// TIA Portal V17 export
// export: Created 2024-09-27T19:06:40.5718073Z, ExportSetting WithDefaults, DisplayName Totally Integrated Automation Portal, DisplayVersion V17, DisplayName TIA Portal Openness, DisplayVersion V17, DisplayName TIA Portal Version Control Interface, DisplayVersion V17, DisplayName STEP 7 Professional, DisplayVersion V17, DisplayName STEP 7 Safety, DisplayVersion V17, DisplayName WinCC Professional, DisplayVersion V17
ORGANIZATION_BLOCK "Main"   // OB1, LAD, ProgramCycle
TITLE = "Main Program Sweep (Cycle)"
{ S7_Optimized_Access := 'TRUE' }
VERSION : 0.1
// stored: AutoNumber true, IsIECCheckEnabled false, SetENOAutomatically false
   VAR_INPUT
      Initial_Call : Bool;   // Initial call of this OB
      Remanence : Bool;   // =True, if remanent data are available
   END_VAR
BEGIN

REGION Network 1: AUTO MODE SET FROM HMI
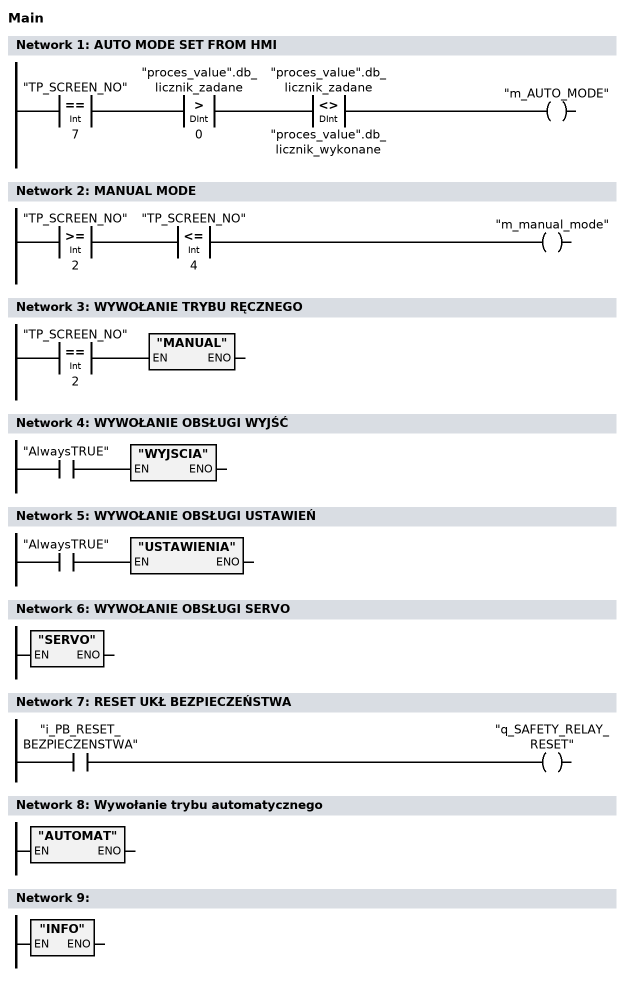
   RUNG wire#powerrail
      { S7_Templates := "SrcType := Int" } EQ_Contact(in1 := "TP_SCREEN_NO", in2 := 7)
      { S7_Templates := "SrcType := DInt" } GT_Contact(in1 := "proces_value".db_licznik_zadane, in2 := 0)
      { S7_Templates := "SrcType := DInt" } NE_Contact(in1 := "proces_value".db_licznik_zadane, in2 := "proces_value".db_licznik_wykonane)
      Coil( "m_AUTO_MODE" )
   END_RUNG
   // the same network as SCL:
   "m_AUTO_MODE" := ("TP_SCREEN_NO" = 7) AND ("proces_value".db_licznik_zadane > 0) AND ("proces_value".db_licznik_zadane <> "proces_value".db_licznik_wykonane);
END_REGION

REGION Network 2: MANUAL MODE
   RUNG wire#powerrail
      { S7_Templates := "SrcType := Int" } GE_Contact(in1 := "TP_SCREEN_NO", in2 := 2)
      { S7_Templates := "SrcType := Int" } LE_Contact(in1 := "TP_SCREEN_NO", in2 := 4)
      Coil( "m_manual_mode" )
   END_RUNG
   // the same network as SCL:
   "m_manual_mode" := ("TP_SCREEN_NO" >= 2) AND ("TP_SCREEN_NO" <= 4);
END_REGION

REGION Network 3: WYWOŁANIE TRYBU RĘCZNEGO
   RUNG wire#powerrail
      { S7_Templates := "SrcType := Int" } EQ_Contact(in1 := "TP_SCREEN_NO", in2 := 2)
      "MANUAL"()
   END_RUNG
   // the same network as SCL:
   IF "TP_SCREEN_NO" = 2 THEN "MANUAL"(); END_IF;
END_REGION

REGION Network 4: WYWOŁANIE OBSŁUGI WYJŚĆ
   RUNG wire#powerrail
      Contact( "AlwaysTRUE" )
      "WYJSCIA"()
   END_RUNG
   // the same network as SCL:
   IF "AlwaysTRUE" THEN "WYJSCIA"(); END_IF;
END_REGION

REGION Network 5: WYWOŁANIE OBSŁUGI USTAWIEŃ
   RUNG wire#powerrail
      Contact( "AlwaysTRUE" )
      "USTAWIENIA"()
   END_RUNG
   // the same network as SCL:
   IF "AlwaysTRUE" THEN "USTAWIENIA"(); END_IF;
END_REGION

REGION Network 6: WYWOŁANIE OBSŁUGI SERVO
   RUNG wire#powerrail
      "SERVO"()
   END_RUNG
   // the same network as SCL:
   "SERVO"();
END_REGION

REGION Network 7: RESET UKŁ BEZPIECZEŃSTWA
   RUNG wire#powerrail
      Contact( "i_PB_RESET_BEZPIECZENSTWA" )
      Coil( "q_SAFETY_RELAY_RESET" )
   END_RUNG
   // the same network as SCL:
   "q_SAFETY_RELAY_RESET" := "i_PB_RESET_BEZPIECZENSTWA";
END_REGION

REGION Network 8: Wywołanie trybu automatycznego
   RUNG wire#powerrail
      "AUTOMAT"()
   END_RUNG
   // the same network as SCL:
   "AUTOMAT"();
END_REGION

REGION Network 9
   RUNG wire#powerrail
      "INFO"()
   END_RUNG
   // the same network as SCL:
   "INFO"();
END_REGION
END_ORGANIZATION_BLOCK
